Staubli VAL3: BackHome.pgx

program BackHome(joint x_jJoint, tool x_tTool, mdesc x_mMdesc, bool& x_bOK)
  local bool l_bHomeOK
  local jointRx l_jJoint
begin
  //-----------------------------------------------------------------------
  //Header begin
  //Description of program
  //  手臂回零，手动模式有效
  //Input parameters
  //  joint  x_jJoint:关节位置；
  //  tool  x_tTool:工具值；
  //  Mdesc x_mMdesc:速度；
  //
  //Output paramaters
  //  bool x_bOK:手臂是否到达零位
  //Example
  //  call AlignPage(tool)
  //History
  //  Creation : 2012-06-11 - PF.Zhong
  //Header end
  //-----------------------------------------------------------------------
  resetMotion()
  x_bOK=false
  if !isPowered()
    popUpMsg("机器人没有上电")
  endIf
  if workingMode()!=1
    popUpMsg("切换到手动模式,并上电")
  endIf
  wait(isPowered() and workingMode()==1)
  l_jJoint=herej()
  if nAxisNum==4 or nAxisNum==6
    call CompareJoint(x_jJoint,l_jJoint,l_bHomeOK,nAxisNum)
    if !l_bHomeOK
      if abs(x_jJoint)<{0.1,0.1,0.1,0.1,0.1,0.1}
        popUpMsg("关节点太接近手臂零点!")
        return
      else
        movej(x_jJoint,x_tTool,x_mMdesc)
        waitEndMove()
        l_jJoint=herej()
        call CompareJoint(x_jJoint,l_jJoint,l_bHomeOK,nAxisNum)
        if l_bHomeOK
          x_bOK=true
        endIf
      endIf
    else
      x_bOK=true
    endIf
  else
    popUpMsg("请输入正确的关节数目!")
    x_bOK=false
  endIf
end
